(* Schneider Machine Expert - Basic project Questao3.5_FelipeV1_20241009, file version 2.9.0.0 *)
(* ProjectInformations: Name=Novo projeto *)

HARDWARE
  Cpu 0: TM221M16R/G
  EthernetConfiguration: NetworkName=M221, IpAllocationMode=FixedAddress, IpAddress=0.0.0.0, SubnetMask=0.0.0.0
  SerialLineConfiguration: Baud=Baud19200, Parity=ParityEven, DataBits=DataBits8, StopBits=StopBits1, PhysicalMedium=PhysicalMediumRs485, TransmissionMode=TransmissionModeModbusRtu, SlaveId=1, Addressing=SlaveAddressing
  MastTask: UsePeriodScanMode=false, PeriodScan=100
  FastTask: Period=255
  CpuBehavior: StartingMode=StartAsPreviousState, AutoSaveRamOnEeprom=true, WatchdogPeriod=250

SYMBOLS  (address, symbol, comment, settings)

POU Entradas
  (* SectionNumber=1 *)

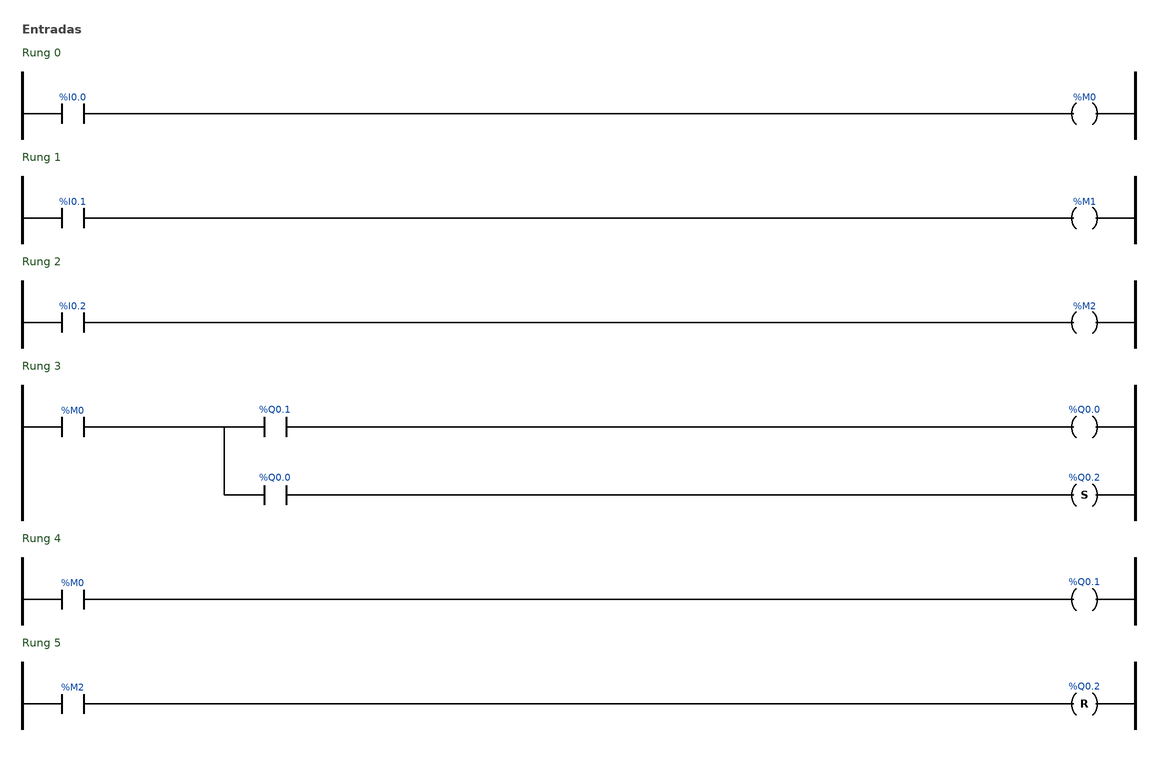

// Rung 0
  LD %I0.0
  ST %M0
  // as ST:
  //   %M0 := %I0.0;

// Rung 1
  LD %I0.1
  ST %M1
  // as ST:
  //   %M1 := %I0.1;

// Rung 2
  LD %I0.2
  ST %M2
  // as ST:
  //   %M2 := %I0.2;

// Rung 3
  LD %M0
  MPS
  AND %Q0.1
  ST %Q0.0
  MPP
  AND %Q0.0
  S %Q0.2
  // as ST:
  //   %Q0.0 := %M0 AND %Q0.1;
  //   IF %M0 AND %Q0.0 THEN %Q0.2 := TRUE; END_IF;

// Rung 4
  LD %M0
  ST %Q0.1
  // as ST:
  //   %Q0.1 := %M0;

// Rung 5
  LD %M2
  R %Q0.2
  // as ST:
  //   IF %M2 THEN %Q0.2 := FALSE; END_IF;
